{attribute 'qualified_only'}
VAR_GLOBAL CONSTANT
	cSizeOfErrorData : UINT := 4;
	
END_VAR

(* stored: Version 1.1.0.1, ProductVersion 3.1.4022.6
   GVL GVL_ErrorSystem: Id {7f2dfaa6-e4ea-4ad1-ac0d-e75f78e9d4ec} *)
